PROGRAM MAIN
VAR	
	// FB_ReadTc3Events
	fbReadTc3Events	   : FB_ReadTc3Events2;
	bReadEvents		   : BOOL							   := TRUE;
	nLanguage		   : DINT							   := 1033;
	eDateAndTimeFormat : Tc2_Utilities.E_DateAndTimeFormat := Tc2_Utilities.E_DateAndTimeFormat.en_US;
	bClearDisplay	   : BOOL;
	eSeverityMin	   : TcEventSeverity;
	bError			   : BOOL;
	hr				   : HRESULT;
	numOfEvents		   : UDINT;
END_VAR

// Call fbReadTc3Events
fbReadTc3Events(bReadEvents		   := bReadEvents,
				nLanguageID		   := nLanguage,
				eDateAndTimeFormat := eDateAndTimeFormat,
				bClearTable		   := bClearDisplay,
				eMinSeverity	   := eSeverityMin,
				nNumberOfEvents	   => numOfEvents,
				bError			   => bError,
				hrErrorCode		   => hr);

bClearDisplay := FALSE;

END_PROGRAM

(* stored: Version 1.1.0.1
   POU MAIN: Id {8e279f0e-7f0a-4414-b3f0-94b367b48d58}, SpecialFunc None *)
